FUNCTION_BLOCK ReactorAvCtrl (* CAT Function Block Type *)
  (* Standard: 61499-2 *)
  (* Version 0.0, 7/15/2026, Schneider Electric, template *)
  PACKAGE SE.Nereda;
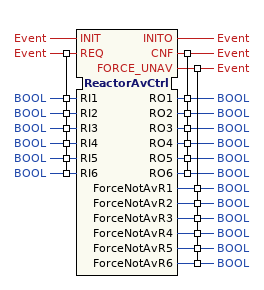
  EVENT_INPUT
    INIT;
    REQ WITH RI1, RI2, RI3, RI4, RI5, RI6; (* Normal Execution Request *)
  END_EVENT
  EVENT_OUTPUT
    INITO;
    CNF WITH RO1, RO2, RO3, RO4, RO5, RO6; (* Execution Confirmation *)
    FORCE_UNAV WITH ForceNotAvR1, ForceNotAvR2, ForceNotAvR3, ForceNotAvR4, ForceNotAvR5, ForceNotAvR6;
  END_EVENT
  VAR_INPUT
    RI1 : BOOL;
    RI2 : BOOL;
    RI3 : BOOL;
    RI4 : BOOL;
    RI5 : BOOL;
    RI6 : BOOL;
  END_VAR
  VAR_OUTPUT
    RO1 : BOOL;
    RO2 : BOOL;
    RO3 : BOOL;
    RO4 : BOOL;
    RO5 : BOOL;
    RO6 : BOOL;
    ForceNotAvR1 : BOOL;
    ForceNotAvR2 : BOOL;
    ForceNotAvR3 : BOOL;
    ForceNotAvR4 : BOOL;
    ForceNotAvR5 : BOOL;
    ForceNotAvR6 : BOOL;
  END_VAR
  FBS
    Reactor1 : SELECT_81F91C08E00C8B28(IN2 := FALSE); {SET_ATTRIBUTE(Configuration.GenericFBType.InterfaceParams, Runtime.Standard#CNT:=2;SELECT:BOOL;IN${CNT$}:BOOL)}
    Reactor2 : SELECT_81F91C08E00C8B28(IN2 := FALSE); {SET_ATTRIBUTE(Configuration.GenericFBType.InterfaceParams, Runtime.Standard#CNT:=2;SELECT:BOOL;IN${CNT$}:BOOL)}
    Reactor3 : SELECT_81F91C08E00C8B28(IN2 := FALSE); {SET_ATTRIBUTE(Configuration.GenericFBType.InterfaceParams, Runtime.Standard#CNT:=2;SELECT:BOOL;IN${CNT$}:BOOL)}
    Reactor4 : SELECT_81F91C08E00C8B28(IN2 := FALSE); {SET_ATTRIBUTE(Configuration.GenericFBType.InterfaceParams, Runtime.Standard#CNT:=2;SELECT:BOOL;IN${CNT$}:BOOL)}
    Reactor5 : SELECT_81F91C08E00C8B28(IN2 := FALSE); {SET_ATTRIBUTE(Configuration.GenericFBType.InterfaceParams, Runtime.Standard#CNT:=2;SELECT:BOOL;IN${CNT$}:BOOL)}
    Reactor6 : SELECT_81F91C08E00C8B28(IN2 := FALSE); {SET_ATTRIBUTE(Configuration.GenericFBType.InterfaceParams, Runtime.Standard#CNT:=2;SELECT:BOOL;IN${CNT$}:BOOL)}
    IThis : ReactorAvCtrl_HMI(QI := TRUE);
  END_FBS
  EVENT_CONNECTIONS
    REQ TO Reactor1.REQ;
    Reactor1.CNF TO Reactor2.REQ;
    Reactor2.CNF TO Reactor3.REQ;
    Reactor3.CNF TO Reactor4.REQ;
    Reactor4.CNF TO Reactor5.REQ;
    Reactor5.CNF TO Reactor6.REQ;
    Reactor6.CNF TO CNF;
    INIT TO IThis.2EB11FFFF95BE31B;
    REQ TO IThis.2CCBFC14FAEC9ED6;
    IThis.6EED28B94E535DE1 TO INITO;
    IThis.0C2C5745E96E6E2C TO Reactor1.REQ;
    IThis.0C2C5745E96E6E2C TO FORCE_UNAV;
  END_CONNECTIONS
  DATA_CONNECTIONS
    Reactor1.OUT TO RO1;
    Reactor2.OUT TO RO2;
    Reactor3.OUT TO RO3;
    Reactor4.OUT TO RO4;
    Reactor5.OUT TO RO5;
    Reactor6.OUT TO RO6;
    RI1 TO Reactor1.IN1;
    RI2 TO Reactor2.IN1;
    RI3 TO Reactor3.IN1;
    RI4 TO Reactor4.IN1;
    RI5 TO Reactor5.IN1;
    RI6 TO Reactor6.IN1;
    RI1 TO IThis.1BF8FC10187018A1;
    RI2 TO IThis.67172E7C4154BBFE;
    RI3 TO IThis.8ED43B091B009467;
    RI4 TO IThis.A93B79CEA845F377;
    RI5 TO IThis.89069F1959C65C18;
    RI6 TO IThis.A66CA3B2FC0B0B19;
    IThis.9DBD772D11E481E7 TO Reactor1.SELECT;
    IThis.A4C40F3EC7F5B963 TO Reactor2.SELECT;
    IThis.886241D9CF0232D7 TO Reactor3.SELECT;
    IThis.40336E0622FF3D72 TO Reactor4.SELECT;
    IThis.C1F4E601C3AC52AA TO Reactor5.SELECT;
    IThis.5AD761AAC6096600 TO Reactor6.SELECT;
    IThis.9DBD772D11E481E7 TO ForceNotAvR1;
    IThis.A4C40F3EC7F5B963 TO ForceNotAvR2;
    IThis.886241D9CF0232D7 TO ForceNotAvR3;
    IThis.40336E0622FF3D72 TO ForceNotAvR4;
    IThis.C1F4E601C3AC52AA TO ForceNotAvR5;
    IThis.5AD761AAC6096600 TO ForceNotAvR6;
  END_CONNECTIONS
END_FUNCTION_BLOCK
